FUNCTION_BLOCK DigitalInput EXTENDS Automation.InputDevice<0>
VAR_INPUT
	SimulatedContactValue : BOOL;
END_VAR
VAR_OUTPUT
	ContactType : CONTACT_TYPE;
END_VAR
VAR
	_ClassName : STRING := __POUNAME();
	
	_CurrentValue : BOOL;
	_PreviousValue : BOOL;
	
	_PhysicalContactValue AT %I* : BOOL;
END_VAR

{attribute 'monitoring' := 'call'}
PROPERTY FINAL Changed : BOOL
GET
Changed := _CurrentValue <> _PreviousValue;
END_GET
END_PROPERTY

{attribute 'monitoring' := 'call'}
PROPERTY ClassName : STRING
GET
ClassName := _ClassName;
END_GET
END_PROPERTY

METHOD FB_init : BOOL
VAR_INPUT
	(* if TRUE, the retain variables are initialized (warm start / cold start)*)
	bInitRetains	: BOOL;
	(* if TRUE, the instance afterwards gets moved into the copy code (online change)*)
	bInCopyCode	: BOOL;
	parent : ISimulatable;
	contactType : CONTACT_TYPE;
END_VAR
THIS^.ContactType := contactType;
END_METHOD

METHOD PROTECTED OnUpdateStateFromInputs
VAR_IN_OUT CONSTANT
	executionContext : Automation.AUTOMATION_EXECUTION_CONTEXT;
END_VAR
_PreviousValue := _CurrentValue;

IF NOT SimulationMode THEN
	_CurrentValue  := _PhysicalContactValue;
ELSE
	_CurrentValue := SimulatedContactValue;
END_IF
END_METHOD

{attribute 'monitoring' := 'call'}
PROPERTY Size : ULINT
GET
Size := XSIZEOF(THIS^);
END_GET
END_PROPERTY

{attribute 'monitoring' := 'call'}
PROPERTY SubDevices : REFERENCE TO ARRAY [0.._SubDeviceCount_ - 1] OF IDevice
GET
SubDevices REF= 0;
END_GET
END_PROPERTY

{attribute 'monitoring' := 'call'}
PROPERTY Value : BOOL
GET
Value := _CurrentValue;
END_GET
END_PROPERTY

END_FUNCTION_BLOCK

(* stored: Version 1.1.0.1
   POU DigitalInput: Id {c6d1eaf1-9cc8-4dbf-a584-1b04597f0f65}, SpecialFunc None
   Property Changed: Id {25fa1762-2c5f-4829-a6e8-7bee560cce1e}
   Get Get: Id {7ff589e4-c33f-4f73-855a-49a7e43cb387}
   Property ClassName: Id {e5420b88-e83e-4617-b101-8fff6688087b}
   Get Get: Id {6468f6c3-92d1-4468-8b70-32b585af0c9f}
   Method FB_init: Id {d6d7f4a6-2485-4546-824a-f61a4f1819bb}
   Method OnUpdateStateFromInputs: Id {a81a5dea-7159-42ed-89a9-6235f07de71d}
   Property Size: Id {3cc9639a-e2ec-49ce-8c2d-d08927803438}
   Get Get: Id {cad1d82f-8f76-41da-8b67-afbeb31a8e85}
   Property SubDevices: Id {a398f56b-2879-48ed-b63b-55852699aa84}
   Get Get: Id {9f77cf10-bd60-44ac-a88c-6f62069bc869}
   Property Value: Id {435debbb-bc61-4a95-9bd6-b412ba0f938a}
   Get Get: Id {5d93ee31-a76c-4b10-880a-8a0871008a6c} *)
